{attribute 'GeneratedUsingTerminal: KL9528'}
{attribute addProperty BoxType "KL9528"}
{attribute addProperty Id "Channel_1AT %Q*Channel_0029832E0"}
{attribute addProperty CRC "2358789635"}
{attribute addProperty Size "0"}
TYPE KL9528_8C984603 :
STRUCT
	{attribute addProperty Name "Channel_1"}
	Channel_1 : Channel_0029832E;
END_STRUCT
END_TYPE

(* stored: Version 1.2.0.0, ProductVersion 3.1.4024.9
   DUT KL9528_8C984603: Id {a08db85b-a888-4b34-bc75-704da5659913} *)
